// TIA Portal V18 export
DATA_BLOCK "DataLogCreate_DB"   // DB64
// stored: AutoNumber true, DBAccessibleFromOPCUA true, InstanceOfName DataLogCreate_SFB, OfSystemLibElement DataLogCreate, OfSystemLibVersion 1.0
"DataLogCreate_SFB"
   // VAR_INPUT
   //    REQ : Bool;
   //    Records : UDInt;
   //    Format : UInt;
   //    Timestamp : UInt;
   //    "Name" : Variant;
   // END_VAR
   // VAR_OUTPUT
   //    DONE : Bool;
   //    BUSY : Bool;
   //    ERROR : Bool;
   //    STATUS : Word;
   // END_VAR
   // VAR_IN_OUT
   //    ID : DWord;
   //    Header : Variant;
   //    Data : Variant;
   // END_VAR
BEGIN
END_DATA_BLOCK
